(* IEC 61131-3 sources: AXOpen/src/AXOpen.Cognex.Vision/ctrl/src/AxoDataman/v_6_0_0/TypeStructuresAndEnums, 4 files *)

(* ---- AxoDataman_Config.st ---- *)
USING System.SerDe;

NAMESPACE AXOpen.Cognex.Vision.v_6_0_0_0
    TYPE
        {#ix-attr:[Container(Layout.Stack)]}
        AxoDataman_Config :
        STRUCT
            ContinuousReading : BOOL := FALSE;
            InfoTime : LTIME := LT#2S;
            ErrorTime : LTIME := LT#5S;
        END_STRUCT;
    END_TYPE
END_NAMESPACE

(* ---- AxoDataman_Results.st ---- *)
NAMESPACE AXOpen.Cognex.Vision.v_6_0_0_0
    TYPE
        AxoDataman_Results :
        STRUCT
            Id: UINT;
            Code: UINT;
            Extended: UINT;
            Length : UINT;
            Data : ARRAY[0..245] OF BYTE;
        END_STRUCT;
    END_TYPE
END_NAMESPACE

(* ---- AxoDataman_SignalStates.st ---- *)
NAMESPACE AXOpen.Cognex.Vision.v_6_0_0_0
    TYPE
        {attribute addProperty Name "<#Signal states#>"}
        {#ix-attr:[Container(Layout.Wrap)]}
        AxoDataman_SignalStates :
        STRUCT
            {attribute addProperty Name "<#Trigger enable#>"}
            TriggerEnable 			:	BOOL;
            {attribute addProperty Name "<#Trigger#>"}
            Trigger					:	BOOL;

            {attribute addProperty Name "<#Enable result buffering#>"}
            EnableResultBuffering	:	BOOL;
            {attribute addProperty Name "<#Result acknowledge#>"}
            ResultsAcknowledge		:	BOOL;

            {attribute addProperty Name "<#Trigger ready#>"}
            TriggerReady 		:	BOOL;
            {attribute addProperty Name "<#Trigger acknowledge#>"}
            TriggerAcknowledge 	:	BOOL;
            {attribute addProperty Name "<#Acquiring#>"}
            Acquiring 			:	BOOL;
            {attribute addProperty Name "<#Missed acquisition#>"}
            MissedAcquisition 	:	BOOL;
            {attribute addProperty Name "<#Trigger ID#>"}
            TriggerID 			:	UINT;

            {attribute addProperty Name "<#Decoding#>"}
            Decoding 				:	BOOL;
            {attribute addProperty Name "<#Decode complete#>"}
            DecodeComplete 			:	BOOL;
            {attribute addProperty Name "<#Result buffer overrun#>"}
            ResultsBufferOverrun 	:	BOOL;
            {attribute addProperty Name "<#Results available#>"}
            ResultsAvailable 		:	BOOL;
            {attribute addProperty Name "<#Error detected#>"}
            ErrorDetected 			:	BOOL;

            {attribute addProperty Name "<#Result ID#>"}
            ResultID 				:	UINT;
            {attribute addProperty Name "<#Result code#>"}
            ResultCode  			:	UINT;
            {attribute addProperty Name "<#Result extended#>"}
            ResultExtended  		:	UINT;
            {attribute addProperty Name "<#Result length#>"}
            ResultLength  			:	UINT;

            {attribute addProperty Name "<#Progress: just for debugging#>"}
            Progress      			:	INT;
        END_STRUCT;
    END_TYPE
END_NAMESPACE

(* ---- AxoDataman_Status.st ---- *)
USING AXOpen.Core;
NAMESPACE AXOpen.Cognex.Vision.v_6_0_0_0
    {#ix-attr:[Container(Layout.Stack)]}
    CLASS AxoDataman_Status EXTENDS AXOpen.Components.Abstractions.AxoComponent_Status
        VAR PUBLIC
            ActionDescriptionPlc : STRING[100];
            ErrorDescriptionPlc : STRING[100];
            SignalStatus : AxoDataman_SignalStates;
            ResultDataSize : eAxoDataman_ResultDataSize := eAxoDataman_ResultDataSize#RESULT_DATA_SIZE_INVALID;
            {#ix-attr:[RenderIgnore()]}
            UserDataSize : eAxoDataman_UserDataSize := eAxoDataman_UserDataSize#USER_DATA_SIZE_INVALID;
        END_VAR
    END_CLASS
END_NAMESPACE
